RoboDK station: NewNozzle.rdk

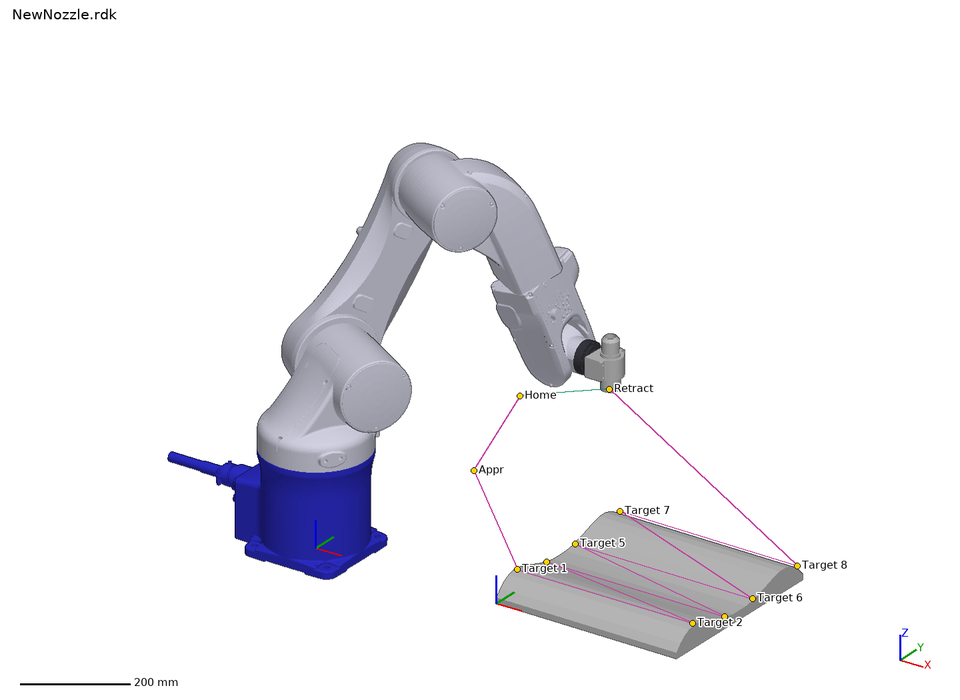
[picture v0: the station drawn from its stored meshes, robots at their saved joint values, targets as dots, program paths as lines]
Station NewNozzle (saved by RoboDK 5.5.4). Poses are relative to the parent item; angles as X-Y-Z fixed-axis rotations.
  - frame Denso VS-6577G-B Base at (0, 0, 0) mm
    - robot Denso VS-6577G-B: 6 axes, payload 7 kg, reach 854 mm, repeatability 0.03 mm, weight 36 kg
        modified DH rows (alpha deg, a mm, theta deg, d mm): 0, 0, 0, 335; -90, 75, -90, 0; 0, 365, -90, 0; -90, 90, 0, 405; 90, 0, 0, 0; -90, 0, 0, 80
        joint limits [-170, -100, -119, -190, -120, -360] to [170, 135, 169, 190, 120, 360]; home [0, 0, 90, 0, 0, 0]; saved at [59.281, 30.207, 128.689, 62.174, -79.795, -18.557]
      - tool NCRDK, TCP at (-50, 0, 30) mm, size 57.1 x 107.2 x 69.8 mm, geometry from NCRDK.STL
      - tool Paint gun, TCP at (40, -10, 450) mm, rotated rx 0 ry 25 rz 0 deg, size 203.2 x 279.7 x 471.5 mm
  - frame Frame 2 at (400, 0, 0) mm
    - object Object Inspection at (0, 0, 0) mm, size 400 x 400 x 46.2 mm, geometry from Object Inspection.stp
    - target Home (Cartesian target) at (56.03, -4.18, 436.99) mm, rotated rx 180 ry -75.55 rz -1.22 deg; joints [-0.222, 17.344, 109.456, 2.533, -22.367, -2.094] of Denso VS-6577G-B
    - target Appr (Cartesian target) at (-49.38, 0.19, 255.02) mm, rotated rx 0 ry -90 rz 178.78 deg; joints [0.425, 16.045, 153.084, 1.672, -79.134, -0.315] of Denso VS-6577G-B
    - target Target 1 (Cartesian target) at (4.23, 62, 45) mm, rotated rx 0 ry -90 rz 178.78 deg; joints [12.333, 63.565, 143.001, 15.08, -115.771, 6.682] of Denso VS-6577G-B
    - target Target 2 (Cartesian target) at (392.83, 62, 45) mm, rotated rx 0 ry -90 rz 178.78 deg; joints [5.382, 76.324, 78.064, 7.311, -64.569, -3.153] of Denso VS-6577G-B
    - target Target 3 (Cartesian target) at (3.09, 155, 23) mm, rotated rx 0 ry -90 rz 178.78 deg; joints [28.226, 66.478, 136.747, 31.559, -110.085, 11.911] of Denso VS-6577G-B
    - target Target 4 (Cartesian target) at (398, 155, 23) mm, rotated rx 0 ry -90 rz 178.78 deg; joints [12.881, 81.609, 70.374, 15.88, -62.898, -7.385] of Denso VS-6577G-B
    - target Target 5 (Cartesian target) at (4, 245, 23) mm, rotated rx 0 ry -90 rz 178.78 deg; joints [40.071, 65.344, 130.294, 42.362, -101.686, 10.465] of Denso VS-6577G-B
    - target Target 6 (Cartesian target) at (398, 245, 23) mm, rotated rx 0 ry -90 rz 178.78 deg; joints [19.773, 84.943, 62.744, 24.416, -60.061, -12.765] of Denso VS-6577G-B
    - target Target 7 (Cartesian target) at (4, 387, 33) mm, rotated rx 0 ry -90 rz 178.78 deg; joints [52.94, 64.933, 116.159, 54.162, -90.639, 0.885] of Denso VS-6577G-B
    - target Target 8 (Cartesian target) at (398, 387, 33) mm, rotated rx 0 ry -90 rz 178.78 deg; joints [29.504, 95.09, 39.401, 40.297, -52.175, -27.476] of Denso VS-6577G-B
    - target Retract (Cartesian target) at (-40.52, 417.56, 255.02) mm, rotated rx 0 ry -90 rz 178.78 deg; joints [50.227, 35.923, 118.298, 54.332, -74.273, -20.69] of Denso VS-6577G-B
  - program ApproachMove (4 instructions, listed below)
  - program MoveTop (10 instructions, listed below)
  - program Retract (4 instructions, listed below)
  - program MainProgram (13 instructions, listed below)
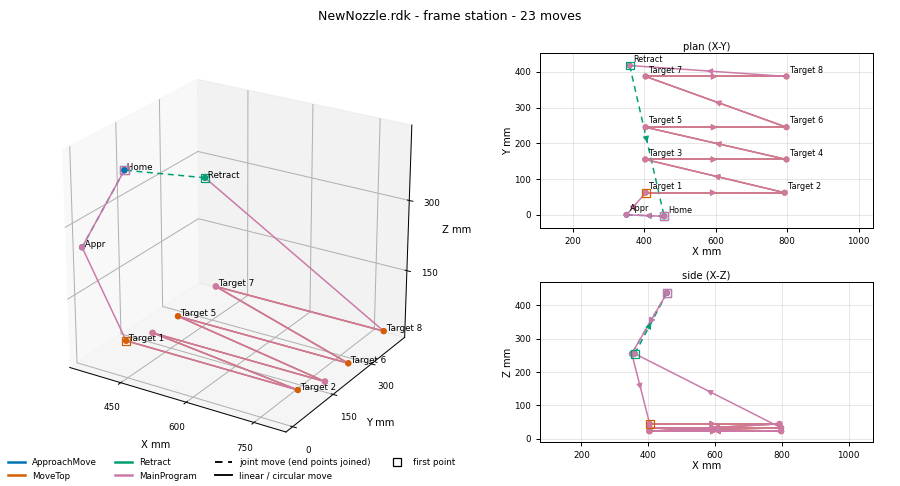
[picture p0: tool path of NewNozzle.rdk in frame station, 23 of 23 moves have a stored position in this frame; points joined in program order, loops and branches not executed]

--- program ApproachMove (robot Denso VS-6577G-B) ---
  Set Ref.: Frame 2
  Set Tool: NCRDK
  MoveJ (Home)
  MoveJ (Appr)

--- program MoveTop (robot Denso VS-6577G-B) ---
  Set Ref.: Frame 2
  Set Tool: NCRDK
  MoveL (Target 1)
  MoveL (Target 2)
  MoveL (Target 3)
  MoveL (Target 4)
  MoveL (Target 5)
  MoveL (Target 6)
  MoveL (Target 7)
  MoveL (Target 8)

--- program Retract (robot Denso VS-6577G-B) ---
  Set Ref.: Frame 2
  Set Tool: NCRDK
  MoveL (Retract)
  MoveJ (Home)

--- program MainProgram (robot Denso VS-6577G-B) ---
  Set Ref.: Frame 2
  Set Tool: NCRDK
  MoveJ (Home)
  MoveL (Appr)
  MoveL (Target 1)
  MoveL (Target 2)
  MoveL (Target 3)
  MoveL (Target 4)
  MoveL (Target 5)
  MoveL (Target 6)
  MoveL (Target 7)
  MoveL (Target 8)
  MoveL (Retract)
